// TwinCAT 3 PLC project PLC1
// Title: HAL
// Company: none
// Author: Tobias Freyermuth
// ProjectVersion: 0.1.0
// Description: Hardware Abstraction Layer of TwinCAT fieldbus devices
// ProgramVersion: 3.1.4024.12
// libraries:
//   Tc2_Standard, * (Beckhoff Automation GmbH)
//   Tc2_System, * (Beckhoff Automation GmbH)
//   Tc3_Module, * (Beckhoff Automation GmbH)
// project tree:
//   / PlcTask.TcTTO (not stored)
//   POUs/ MAIN.TcPOU
//   Project Information/ F_GetCompany.TcPOU (not stored), F_GetTitle.TcPOU, F_GetVersion.TcPOU (not stored)
//   Version/ Global_Version.TcGVL (not stored)

// ---- POUs/MAIN.TcPOU
PROGRAM MAIN
VAR
END_VAR

END_PROGRAM

// ---- Project Information/F_GetTitle.TcPOU
// This function has been automatically generated from the project information.
{attribute 'signature_flag' := '1073741824'}
{attribute 'TcGenerated'}
{attribute 'no-analysis'}
FUNCTION F_GetTitle : WSTRING
VAR_INPUT
	
END_VAR

F_GetTitle := "HAL";

END_FUNCTION
